(* IEC 61131-3 sources: mect_apps/TPAC1006/Collaudo_PLC, 6 files *)

(* ---- LIO_TPAC1007.gvl ---- *)
(* Global variable file *)
VAR_GLOBAL

	(* Local Input Output variables TPAC1007 *)

 	   	TP1007_LIO_Revision AT %IW5.00: UINT;

		TP1007_LIO_DigDir_1_8 AT %QB5.04: BYTE;
		TP1007_LIO_DigDir_1 AT %QX5.04.0: BOOL;
		TP1007_LIO_DigDir_2 AT %QX5.04.1: BOOL;
		TP1007_LIO_DigDir_3 AT %QX5.04.2: BOOL;
		TP1007_LIO_DigDir_4 AT %QX5.04.3: BOOL;
		TP1007_LIO_DigDir_5 AT %QX5.04.4: BOOL;
		TP1007_LIO_DigDir_6 AT %QX5.04.5: BOOL;
		TP1007_LIO_DigDir_7 AT %QX5.04.6: BOOL;
		TP1007_LIO_DigDir_8 AT %QX5.04.7: BOOL;

		TP1007_LIO_DigIn_1_8 AT %IB5.12: BYTE;
		TP1007_LIO_DigIn_1 AT %IX5.12.0: BOOL;
		TP1007_LIO_DigIn_2 AT %IX5.12.1: BOOL;
		TP1007_LIO_DigIn_3 AT %IX5.12.2: BOOL;
		TP1007_LIO_DigIn_4 AT %IX5.12.3: BOOL;
		TP1007_LIO_DigIn_5 AT %IX5.12.4: BOOL;
		TP1007_LIO_DigIn_6 AT %IX5.12.5: BOOL;
		TP1007_LIO_DigIn_7 AT %IX5.12.6: BOOL;
		TP1007_LIO_DigIn_8 AT %IX5.12.7: BOOL;

		TP1007_LIO_DigOut_1_8 AT %QB5.24: BYTE;
		TP1007_LIO_DigOut_1 AT %QX5.24.0: BOOL;
		TP1007_LIO_DigOut_2 AT %QX5.24.1: BOOL;
		TP1007_LIO_DigOut_3 AT %QX5.24.2: BOOL;
		TP1007_LIO_DigOut_4 AT %QX5.24.3: BOOL;
		TP1007_LIO_DigOut_5 AT %QX5.24.4: BOOL;
		TP1007_LIO_DigOut_6 AT %QX5.24.5: BOOL;
		TP1007_LIO_DigOut_7 AT %QX5.24.6: BOOL;
		TP1007_LIO_DigOut_8 AT %QX5.24.7: BOOL;

		TP1007_LIO_AnIn_1 AT %IW5.14: INT;
		TP1007_LIO_AnIn_2 AT %IW5.16: INT;

		TP1007_LIO_Tamb AT %IW5.18 : INT;
		TP1007_LIO_EncoderLo AT %IW5.20: UINT;
		TP1007_LIO_EncoderHi AT %IW5.22: UINT;

		TP1007_LIO_EncoderEnable AT %QW5.28: WORD;
		TP1007_LIO_EncoderReset AT %QW5.30: WORD;

		TP1007_LIO_AnOut_1 AT %QW5.26: INT;

		(* TP1007_LIO_AnIn_Conf *)
		TP1007_LIO_AnInConf_1 AT %QW5.06: WORD;
		TP1007_LIO_AnInConf_2 AT %QW5.08: WORD;

		(* TP1007_LIO_AnOut_Conf *)
		TP1007_LIO_AnOut_Conf AT %QW5.10: WORD;

		TP1007_LIO_DigIn_9_12 AT %IB5.13: BYTE;
		TP1007_LIO_DigIn_9 AT %IX5.13.0: BOOL;
		TP1007_LIO_DigIn_10 AT %IX5.13.1: BOOL;
		TP1007_LIO_DigIn_11 AT %IX5.13.2: BOOL;
		TP1007_LIO_DigIn_12 AT %IX5.13.3: BOOL;

END_VAR

(* ---- Resource1.gvl ---- *)
(* Global variable file *)
VAR_GLOBAL
RET_AnInConf_1 AT %MW0.4:UINT;
RET_AnInConf_2 AT %MW0.8:UINT;
RET_AnInConf_3 AT %MW0.12:UINT;
RET_AnInConf_4 AT %MW0.16:UINT;
RET_AnOutConf_1 AT %MW0.20:UINT;
RET_AnOutConf_2 AT %MW0.24:UINT;
CAN1_IN_DIG_8_1 AT %MW0.5380:INT;
CAN1_IN_DIG_8_2 AT %MW0.5384:INT;
CAN1_OUT_DIG_8_1 AT %MW0.5388:INT;
CAN1_OUT_DIG_8_2 AT %MW0.5392:INT;
CAN1_IN_AN_1 AT %MW0.5396:INT;
CAN1_IN_AN_2 AT %MW0.5400:INT;
CAN1_IN_AN_3 AT %MW0.5404:INT;
CAN1_IN_AN_4 AT %MW0.5408:INT;
CAN1_IN_AN_5 AT %MW0.5412:INT;
CAN1_IN_AN_6 AT %MW0.5416:INT;
CAN1_IN_AN_7 AT %MW0.5420:INT;
CAN1_IN_AN_8 AT %MW0.5424:INT;
CAN1_IN_AN_9 AT %MW0.5428:INT;
CAN1_IN_AN_10 AT %MW0.5432:INT;
CAN1_IN_AN_11 AT %MW0.5436:INT;
CAN1_IN_AN_12 AT %MW0.5440:INT;
CAN1_IN_AN_13 AT %MW0.5444:INT;
CAN1_IN_AN_14 AT %MW0.5448:INT;
CAN1_IN_AN_15 AT %MW0.5452:INT;
CAN1_IN_AN_16 AT %MW0.5456:INT;
CAN1_OUT_AN_1 AT %MW0.5460:INT;
Modbus_1 AT %MW0.5464:INT;
Parti AT %MW0.5468:INT;
END_VAR

(* ---- fb_HW119_LoadCrossTab.st ---- *)
(*[[
]]*)
FUNCTION_BLOCK fb_HW119_LoadCrossTab
#import "Resource1.gvl"
#import "crosstable.gvl"
VAR_INPUT
	ENABLE:BOOL;		(* Abilitazione funzione*)
	CTFile:STRING;		(* file di cross table da aprire	*)
	CTDimension:DINT;	(* dimensione della cross table da leggere	*)
	CTType:UINT;		(* tipo di cross table da leggere	*)
END_VAR
VAR_OUTPUT
	END:BOOL;			(* Fine funzione	*)
	ERR:BOOL;			(* segnalazione errore	*)
END_VAR
VAR
		InitXtable: fb_HW119_Init;
		ReadFields:fb_HW119_ReadVarFields;
		ReadAlarmsFields:fb_HW119_ReadAlarmsFields;
		ReadCommFields:fb_HW119_ReadCommFields;
		FBState: UINT;
		FunctRes:UINT;
		index: DINT;
		STEPS:DINT:=50;
		LowEdge:DINT:=0;
		HiEdge:DINT:=0;
END_VAR
IF ENABLE THEN
	IF FBState = 0 THEN
		InitXtable(TIPO:=CTType);													(* Inizializzazione delle variabili CT*)
		FBState:=10;
		ErrorsState:=ErrorsState AND 16#F0;											(* reset flag di errore*)
		LowEdge:=1;
		HiEdge:=STEPS;
		IF HiEdge > CTDimension THEN
			HiEdge:=CTDimension;
		END_IF;
	ELSIF FBState =10	THEN												(* OPEN CROSS TABLE*)
		FunctRes:=HW119_OpenCrossTable(CTFile);
		IF FunctRes = 0 THEN												(* Operazione andata a buon fine	*)
			FBState:=20;
			HW119_ERR[2]:=2;
		ELSE
			FBState:=1000;													(* Errore -> termina	*)
			ErrorsState:=ErrorsState OR 16#01;
			HW119_ERR[2]:=3;
		END_IF;

	ELSIF FBState =20	THEN												(* LOAD CROSS TABLE RECORDS*)
		FOR index:=LowEdge TO HiEdge	DO									(* lettura di STEPS record di CT	*)
			IF CTType > 0 	THEN											(* Se CT non è quella delle variabili non si aggiunge alla Hash*)
		 		FunctRes:=HW119_ReadCrossTableRecord(TRUE);					(* LEGGE RECORD DELLA CROSSTABLE*)
			ELSE
				FunctRes:=HW119_ReadCrossTableRecord(FALSE);				(* LEGGE RECORD DELLA CROSSTABLE lo aggiunge alla HAsh*)
			END_IF;

			IF FunctRes = 0 THEN
				HW119_ERR[1]:=2;
				CASE CTType OF
					0:		ReadFields(Index:=DINT_TO_INT(index));			(* lettura crosstable variabili	*)
							IF ReadFields.ERR THEN
								CrossTable[index].Error:=100;				(* marca la entry della crosstable come errata*)
								ErrorsState:=ErrorsState OR 16#04;
							END_IF;
					1:		ReadAlarmsFields(Index:=DINT_TO_INT(index));	(* lettura crosstable Allarmi	*)
							IF ReadAlarmsFields.ERR 	 THEN
								ALCrossTable[index].ALError:=100;			(* marca la entry della crosstable ALLARMI come errata*)
								ErrorsState:=ErrorsState OR 16#04;
							END_IF;
					ELSE
					ReadCommFields(Index:=DINT_TO_INT(index));				(* lettura CT dei parametri di comunicazione	*)
					IF index > 1 	THEN
						IF ReadCommFields.ERR 	THEN
							CommParameters[index-1].State:=FALSE;
						ELSE
							CommParameters[index-1].State:=TRUE;
						END_IF;
					 END_IF;
				END_CASE;
			ELSE
				HW119_ERR[1]:=3;
				IF CTType = 0	 THEN
					CrossTable[index].Error:=100;						(* marca la entry della crosstable come non ancora aggiornata*)
					ErrorsState:=ErrorsState OR 16#02;
				ELSIF CTType = 1	 THEN
					ALCrossTable[index].ALError:=100;					(* marca la entry della crosstable ALLARMI come non ancora aggiornata*)
					ErrorsState:=ErrorsState OR 16#04;
				END_IF;
			END_IF;

		END_FOR;
		FBState:=30;

	ELSIF FBState = 30	THEN
		LowEdge:=HiEdge+1;
		HiEdge:=HiEdge+STEPS;
		IF LowEdge < CTDimension	THEN								(* controlla se è terminata la CT da legere	*)
			IF HiEdge<CTDimension THEN
				FBState:=20;
			ELSIF HiEdge>=CTDimension THEN
				HiEdge:=CTDimension;
				FBState:=20;
			 END_IF;
		ELSE
			FBState:=40;
		END_IF;

	ELSIF FBState = 40	THEN
		FunctRes:=HW119_CloseCrossTable();											(* CLOSE CrossTable*)
		IF FunctRes = 0 THEN
			HW119_ERR[0]:=2;				(*debug*)
		 	FBState:= 100;
		ELSE
			FBState:=1000;
			HW119_ERR[0]:=3;				(*debug*)
			ErrorsState:=ErrorsState OR 16#08;
		END_IF;
	ELSIF FBState = 100	THEN														(* TERMINATA LETTURA CROSSTABLE*)
		END:=TRUE;
	ELSIF FBState = 1000 THEN														(* TERMINATA LETTURA CROSSTABLE*)
		FunctRes:=HW119_CloseCrossTable();											(* CLOSE CrossTable*)
		FBState:= 1010;
		ERR:=TRUE;
	END_IF;
ELSE
	END:=FALSE;
	ERR:=FALSE;
	FBState:= 0;
END_IF;
END_FUNCTION_BLOCK

(* ---- fb_HW119_ReadAlarmsFields.st ---- *)
(*[[
]]*)
FUNCTION_BLOCK fb_HW119_ReadAlarmsFields
#import "Resource1.gvl"
#import "crosstable.gvl"
VAR_INPUT
	Index:INT;
END_VAR
VAR_OUTPUT
	ERR:BOOL;
END_VAR

VAR
	Field:STRING;
	FunctRes:UINT;
END_VAR

	ERR:=FALSE;
	FunctRes:=HW119_GetCrossTableField(Field);				(*Lettura TIPO 0 : evento, 1 : allarme*)
	IF FunctRes = 0 THEN
		ALCrossTable[index].ALType:=STRING_TO_BOOL(Field);
	ELSE
		ERR:=TRUE;
	END_IF;

	FunctRes:=HW119_GetCrossTableField(Field);				(* variabile di allarme	*)
	IF FunctRes = 0 THEN
		ALCrossTable[index].ALTag:=Field;
	ELSE
		ERR:=TRUE;
	END_IF;

	FunctRes:=HW119_GetCrossTableField(Field);				(* Variabile di sorgente	*)
	IF FunctRes = 0 THEN
		ALCrossTable[index].ALSource:=Field;
	ELSE
		ERR:=TRUE;
	END_IF;

	FunctRes:=HW119_GetCrossTableField(Field);				(* variabile di confronto	*)
	IF FunctRes = 0 THEN
		ALCrossTable[index].ALCompareVar:=Field;
	ELSE
		ERR:=TRUE;
	END_IF;

	FunctRes:=HW119_GetCrossTableField(Field);
	IF FunctRes = 0 THEN
		ALCrossTable[index].ALCompareVal:=STRING_TO_DWORD(Field);
	ELSE
		ERR:=TRUE;
	END_IF;

	FunctRes:=HW119_GetCrossTableField(Field);
	IF FunctRes = 0 THEN
		ALCrossTable[index].ALOperator:=STRING_TO_UINT(Field);
	ELSE
		ERR:=TRUE;
	END_IF;

	FunctRes:=HW119_GetCrossTableField(Field);
	IF FunctRes = 0 THEN
		ALCrossTable[index].ALFilterTime:=STRING_TO_UINT(Field);
		ALCrossTable[Index].ALFilterCount:=ALCrossTable[index].ALFilterTime;
	ELSE
		ERR:=TRUE;
	END_IF;

END_FUNCTION_BLOCK

(* ---- PLC.st ---- *)
(*[[
]]*)
PROGRAM PLC
#import "Resource1.gvl"
#import "crosstable.gvl"
#import "TPACLocaIO.gvl" (* <---= *)
#import "Collaudo_CAN.gvl"
#import "LIO_TPAC1006.gvl"
VAR
	fb_HW119_PLCwriteVar_Inst : fb_HW119_PLCwriteVar;
	counter : UDINT := 0;
	divisor : UDINT := 10;
	values : ARRAY [0..15] OF DWORD;
	TIMER1:TON;
	TIMER2:TON;
END_VAR;
if Parti = 1 then
	TIMER2(IN:=TRUE,PT:=T#1s);
	IF TIMER2.Q THEN
	TIMER2(IN:=FALSE,PT:=T#1s);
		if counter = 0 * divisor then
			PLC_DigOut_1:=0;
			PLC_DigOut_2:=0;
			PLC_DigOut_3:=0;
			PLC_DigOut_4:=0;
			PLC_DigOut_5:=0;
			PLC_DigOut_6:=0;
			PLC_DigOut_7:=0;
			PLC_DigOut_8:=0;
			PLC_DigOut_9:=0;
			PLC_DigOut_10:=0;
			PLC_DigOut_11:=0;
			PLC_DigOut_12:=0;
			PLC_DigOut_13:=0;
			PLC_DigOut_14:=0;
			PLC_DigOut_15:=0;
			PLC_DigOut_16:=0;
		elsif counter = 1  then
			PLC_DigOut_1 := 1;
		elsif counter = 2  then
			PLC_DigOut_1 := 0;
			PLC_DigOut_2 := 1;
		elsif counter = 3 then
			PLC_DigOut_2 := 0;
			PLC_DigOut_3 := 1;
		elsif counter = 4 then
			PLC_DigOut_3 := 0;
			PLC_DigOut_4 := 1;
		elsif counter = 5 then
			PLC_DigOut_4 := 0;
			PLC_DigOut_5 := 1;
		elsif counter = 6 then
			PLC_DigOut_5 := 0;
			PLC_DigOut_6 := 1;
		elsif counter = 7 then
			PLC_DigOut_6 := 0;
			PLC_DigOut_7 := 1;
		elsif counter = 8 then
			PLC_DigOut_7 := 0;
			PLC_DigOut_8 := 1;
		elsif counter = 9 then
			PLC_DigOut_8 := 0;
			PLC_DigOut_9 := 1;
		elsif counter = 10 then
			PLC_DigOut_9 := 0;
			PLC_DigOut_10 := 1;
		elsif counter = 11 then
			PLC_DigOut_10 := 0;
			PLC_DigOut_11 := 1;
		elsif counter = 12  then
			PLC_DigOut_11 := 0;
			PLC_DigOut_12 := 1;
		end_if;

		counter := counter + 1;

		if counter > 13  then
			counter := 0;
		end_if;
	end_if;

values[0]:=1;
fb_HW119_PLCwriteVar_Inst(VARIABLE := 'Modbus_1', VALUES := values, Nregs := 1);
IF FALSE THEN
	ch1_CAN1_OUT_DIG_8_1:=0;
END_IF;
TIMER1(in:=TRUE,PT:=T#1s);
IF TIMER1.Q THEN
	TIMER1(in:=FALSE,PT:=T#1s);
	IF ch1_CAN1_OUT_DIG_8_1 = 16#01 THEN
		ch1_CAN1_OUT_DIG_8_1:=16#01;
	ELSE
		ch1_CAN1_OUT_DIG_8_1:=16#00;
	END_IF;
END_IF;
end_if;
PLC_CAN1_IN_AN_1:=ch1_CAN1_IN_AN_1;
PLC_CAN1_IN_AN_2:=ch1_CAN1_IN_AN_2;
PLC_CAN1_IN_AN_3:=ch1_CAN1_IN_AN_3;
PLC_CAN1_IN_AN_4:=ch1_CAN1_IN_AN_4;
PLC_CAN1_IN_AN_5:=ch1_CAN1_IN_AN_5;
PLC_CAN1_IN_AN_6:=ch1_CAN1_IN_AN_6;
PLC_CAN1_IN_AN_7:=ch1_CAN1_IN_AN_7;
PLC_CAN1_IN_AN_8:=ch1_CAN1_IN_AN_8;
PLC_CAN1_IN_AN_9:=ch1_CAN1_IN_AN_9;
PLC_CAN1_IN_AN_10:=ch1_CAN1_IN_AN_10;
PLC_CAN1_IN_AN_11:=ch1_CAN1_IN_AN_11;
PLC_CAN1_IN_AN_12:=ch1_CAN1_IN_AN_12;
PLC_CAN1_IN_AN_13:=ch1_CAN1_IN_AN_13;
PLC_CAN1_IN_AN_14:=ch1_CAN1_IN_AN_14;
PLC_CAN1_IN_AN_15:=ch1_CAN1_IN_AN_15;
PLC_CAN1_IN_AN_16:=ch1_CAN1_IN_AN_16;
if  PLC_AnOutConf_1 <> UINT_TO_WORD(RET_AnOutConf_1)then
	PLC_AnOut_1 := 0;
	PLC_AnOutConf_1 := UINT_TO_WORD(RET_AnOutConf_1);
end_if;
if  PLC_AnOutConf_2 <> UINT_TO_WORD(RET_AnOutConf_2)then
	PLC_AnOut_2 := 0;
	PLC_AnOutConf_2 := UINT_TO_WORD(RET_AnOutConf_2);
end_if;

PLC_AnInConf_1 := UINT_TO_WORD(RET_AnInConf_1);
PLC_AnInConf_2 := UINT_TO_WORD(RET_AnInConf_2);
PLC_AnInConf_3 := UINT_TO_WORD(RET_AnInConf_3);
PLC_AnInConf_4 := UINT_TO_WORD(RET_AnInConf_4);

(* limits the overflow value *)
IF (INT_TO_WORD(TP1006_LIO_AnOut_Conf) AND 16#01) = 16#01 THEN
	IF PLC_AnOut_1 > 2000 then
		PLC_AnOut_1:=2000;
	END_IF;
	IF PLC_AnOut_1 < 0 then
		PLC_AnOut_1:=0;
	END_IF;
END_IF;
IF (INT_TO_WORD(TP1006_LIO_AnOut_Conf) AND 16#02) = 16#02 THEN
	IF PLC_AnOut_1 > 1000 then
		PLC_AnOut_1:=1000;
	END_IF;
	IF PLC_AnOut_1 < 0 then
		PLC_AnOut_1:=0;
	END_IF;
END_IF;
IF (INT_TO_WORD(TP1006_LIO_AnOut_Conf) AND 16#10)  = 16#10 THEN
	IF PLC_AnOut_2 > 2000 then
		PLC_AnOut_2:=2000;
	END_IF;
	IF PLC_AnOut_2 < 0 then
		PLC_AnOut_2:=0;
	END_IF;
END_IF;
IF (INT_TO_WORD(TP1006_LIO_AnOut_Conf) AND 16#20)  = 16#20 THEN
	IF PLC_AnOut_2 > 1000 then
		PLC_AnOut_2:=1000;
	END_IF;
	IF PLC_AnOut_2 < 0 then
		PLC_AnOut_2:=0;
	END_IF;
END_IF;
END_PROGRAM

(* ---- Program1.st ---- *)
(*[[
    UserHelpURL= "4cfile:Program1.HTML",
]]*)

PROGRAM Program1
#import "crosstable.gvl"
VAR
(* Revisione 5.31
Corretto baco nel blocco funzione PLCsync
riga 35					FOR I:=0 TO CrossTable[addr].NReg-1 BY STEPS DO
aggiunto -1 al FOR
*)

(* Revisione 5.32
Inserita la misurazione della query pause al termine della risposta dallo slave
solo per protocollo RTU
*)

(* Revisione 5.33
Modificata policy del device disconnesso. Ora, se un indirizzo non risponde e supera il limite faildivisor
si mette l'indirizzo in una blacklist, quindi le richieste di accessi successivi al device saranno ignorati

Revisione 5.4
Inseriti contatori di errori per ogni protocollo
	ContatoreErroriRTU
	ContatoreErroriTCP
	ContatoreErroriTCPRTU

Inserite variabili di revisione:
	PLCRevision01
	PLCRevision02

Modificata scrittura in uPLC: Le scritture sono prioritarie rispetto a quelle HMI, sono ammesse le scritture multiple
Inserita la gestione delle variabili intere a 32 bit
	UDINTDCBA
	UDINTCDAB
	UDINTABCD
	UDINTBADC
	DINTDCBA
	DINTCDAB
	DINTABCD
	DINTBADC

 Revisione 5.42
 	Inserite scritture ad alta priorità da uPLC
	Le scritture sono inserite in tre code (una per protocollo) ed eseguite nella sequenza di arrivo
	tutte le altre operazioni sono ritardate fino a che non sono
	terminate le scritture

Revisione 5.43
	Corretto baco già risolto in 5.31, reintrodotto nella 5.4.
Revisione 5.44
	Corretto baco sulla gestione allarmi: Non veniva effettuato l'aggiornamento dello stato della variabile a error=0
		nel caso di accessi interni (non su strumenti) sia da HMI che da uPLC
		Perciò se la SourceVariable era una variabile interna (non su un device modbus)
		non veniva aggiornato lo stato di variabile disponibile per gli allarmi
		corretto file PLC_sync.st
		aggiunta alla riga 35 CrossTable[addr+I].Error:=0;
	Corretto baco sulle scritture da PLC:
		non venivano effettuate le scritture multiple se il uPLC le effettuava su variabili interne
		modificato nel blocco funzione fb_HW119_PLCwriteVar il codice
					FOR I:=0 TO NRegs-1 DO
						ARRAY_CROSSTABLE_INPUT[WORD_TO_INT(ADDRESS)+I]:=CrossTable[WORD_TO_INT(ADDRESS)+I].PLCWriteVal;
						CrossTable[WORD_TO_INT(ADDRESS)+I].Error:=0;
					END_FOR;
Revisione 5.45
	Corretto baco su scritture multiple

Revisione 5.46
	Corretto baco su scritture singole

Revisione 5.47
	Modificata gestione ricetta
	Aggiunta scrittura in ricetta delle variabili interne

Revisione 5.48
	Corretta la gestione dei falg di busywrite per le scritture su variabili interne nel blocco funzione PLCsync
Revisione 5.49
	Corretto baco su FB plcsync: non veniva aggiornata la mandata in run del protocollo TCP a seguito di una riconnessione
Revisione 5.50
	Corretta letura Modbus sui bit nei protocolli RTU e TCPRTU
Revisione 5.51
	Corretta la gestione della scrittura a bit da PLC interno
	Corretta la segnalazione di errore nel blocco funzione fb_HW119_PLCwriteVar
	MOdificato blocco fb_HW119_AlarmsMngr: in caso di variabili interne non si controlla se è già avvenuta l'assegnazione
Revisione 5.52
	Corretta gestione fb_HW119_PLCwritevar in caso di errore sulla funzione Gettaddr()
Revisione 5.53
	Aggiunta scrittura multipla delle variabili interne
Revisione 6.00
	Inserita priorità delle letture
	contatori errore e blacklist
	scritture ad interrupt
Revisione 6.01
	Corretti bachi:
		La variabile Retry non veniuva azzerata se il dispositivo ritornava on line prima dello scadere dei retry
		messa a false la variabile debug
		corretta la revisione sw
		aggiunta variabilie di Error_flag che segnala se c'è stato almeno un errore dall'ultimo reset
Revisione 6.02
		corretto baco su scrittura da PLC
		aggiunto a Error_flag la segnalazione di errore sulla lettura di una crosstable
Revisione 6.03
		modificate costanti dei file delle CT: tolti i path per poter essere utilizzati da SD
		non si tiene conto del  path per le crosstable per il caricamento da Flash o SD card
Revisione 6.04
	Inserito di default NodeId a 1 nel caso di protocollo TCP

Revisione 6.05
	Inserita gestione Canopen in funzione della variabile HardwareType
	variata la gestione delle scritture e letture nel task RTU
Revisione 6.08
	corretti bachi sui protocolli
Revisione 6.10
	corretti bacho su fb_HW119_MODBUS
Revisione 6.12
	Modificati file gvl delle variabili locali
	creato blocco funzione di sincronizzazione per le variabili locali del tpac1007
	unificate le variabili di IO locale PLC di accesso utente
	inserita la variabile di sistema PLC_time per che si azzera ogni 3600 secondi
 Revisione 6.13
 	Modificate uscite analogiche sui blocchi funzione fb_TPAC1006_LIO_sync e fb_TPAC1007_LIO_sync
*)

	InitComm:fb_HW119_InitComm;
	AlarmMngr:fb_HW119_AlarmsMngr;
	LoadXTable:fb_HW119_LoadCrossTab;
	ErrorMNG:fb_HW119_ErrorMng;
	PLCsync:fb_HW119_PLCsync;
	Reconnect:fb_HW119_Check;
	TPAC1006_LIOsync:fb_TPAC1006_LIOsync;
	TPAC1007_LIOsync:fb_TPAC1007_LIOsync;
	TICtimer:fb_TPAC_tic;
	FunctRes:UINT;
	CommState: UDINT;
	COUNTER:UDINT;
	timer_sync:TON;

	(* DEBUG
	errorT1:DINT;
	errorT2:DINT;
	errorT3:DINT;
	errorT4:DINT;
	reterr:WORD;
	*)
END_VAR
(*	DEBUG
	errorT1:=GetLocalTaskErrno ('Task1');
	errorT2:=GetLocalTaskErrno ('Task2_RTU'	);
	errorT3:=GetLocalTaskState ('Task1');
	errorT4:=GetLocalTaskState('Task2_RTU');
	PLCRevision01:=5;
	PLCRevision02:=4;
*)

	IF CommState = 0	THEN
		FunctRes:=HW119_CloseCrossTable();
		LoadXTable(ENABLE:=FALSE);
		InitComm(ENABLE:=FALSE);
		ErrorsState:=0;
		CommState:=10;
		COUNTER:=0;
		RTU_RUN:=FALSE;
		TCP_RUN:=FALSE;
		TCPRTU_RUN:=FALSE;
		ERROR_FLAG:=0;
	ELSIF CommState = 10	THEN			(* Lettura crosstable allarmi	*)
		LoadXTable(ENABLE:=TRUE,CTFile:=ALcrossTableFile,CTDimension:=DimAlarmsCT,CTType:=1);
		IF LoadXTable.ERR  	THEN
			CommState:=20;					(* Fallita lettura crosstable allrmi -> prosegue con lettura cross table variabili*)
			ALCrossTableState:=FALSE;
			LoadXTable(ENABLE:=FALSE);
			ERROR_FLAG:=ERROR_FLAG OR 16#10;(* SEGNALO L'ERRORE SUL BIT 4*)
		ELSE
			IF LoadXTable.END THEN
				CommState:=20;				(*lettura crosstable  Allarmi  OK  -> prosegue*)
				FunctRes:=HW119_CloseCrossTable();
				LoadXTable(ENABLE:=FALSE);
			END_IF;
		END_IF;

	ELSIF CommState = 20	THEN			(* Lettura crosstable variabili	*)
		LoadXTable(ENABLE:=TRUE,CTFile:=VARcrossTableFile,CTDimension:=DimCrossTable,CTType:=0);
		IF LoadXTable.ERR  	THEN
			CommState:=1000;
			CrossTableState:=FALSE;			(* Fallita lettura crosstable  variabili: FINE*)
			ERROR_FLAG:=ERROR_FLAG OR 16#20;(* SEGNALO L'ERRORE SUL BIT 5*)
		ELSE
			IF LoadXTable.END THEN
				CommState:=30;				(*lettura crosstable  variabili  OK ->  prosegue*)
				LoadXTable(ENABLE:=FALSE);
			END_IF;
		END_IF;

	ELSIF CommState = 30	THEN			(* Lettura crosstable parametri di comunicazione	*)
		LoadXTable(ENABLE:=TRUE,CTFile:=CommParFile,CTDimension:=5,CTType:=2);
		IF LoadXTable.ERR  	THEN
			CommState:=1000;				(* Fallita lettura crosstable  parametri di comunicazione: FINE*)
			ERROR_FLAG:=ERROR_FLAG OR 16#08;(* SEGNALO L'ERRORE SUL BIT 3*)
		ELSE
			IF LoadXTable.END THEN
				CommState:=40;				(*lettura crosstable  variabili  OK ->  prosegue*)
				LoadXTable(ENABLE:=FALSE);
			END_IF;
		END_IF;

	(* Abilitazione protocollo RTU se almeno una entry della crosstable supporta questo protocollo*)
	ELSIF CommState = 40	THEN
		IF 	RTUProtocol_ON	AND CommParameters[1].State THEN
			InitComm(ENABLE:=TRUE,Interface:='RTU');	(*inizializza comunicazione	*)
			IF InitComm.END THEN
				FunctRes:=WORD_TO_UINT(TSK_Start('TASK2_RTU'));		(* partenza task RTU*)
				ERROR_FLAG:=ERROR_FLAG OR 16#80;(* SEGNALO CHE IL TASK RTU è PARTITO*)
				CommState:=50;
				InitComm(ENABLE:=FALSE);
				RTU_RUN:=TRUE;
			ELSIF InitComm.ERR THEN
				CommState:=50;
				InitComm(ENABLE:=FALSE);
				RTU_RUN:=FALSE;
			END_IF;
		ELSE
			CommState:=50;
		END_IF;

	(* Abilitazione protocollo TCP se almeno una entry della crosstable supporta questo protocollo*)
	ELSIF CommState = 50	THEN
		IF 	TCPProtocol_ON	AND CommParameters[2].State THEN
			InitComm(ENABLE:=TRUE,Interface:='TCP');	(*inizializza comunicazione	*)
			IF InitComm.END THEN
				FunctRes:=WORD_TO_UINT(TSK_Start('TASK3_TCP'));		(* partenza task TCP*)
				ERROR_FLAG:=ERROR_FLAG OR 16#100;(* SEGNALO CHE IL TASK TCP è PARTITO*)
				CommState:=60;
				InitComm(ENABLE:=FALSE);
				TCP_RUN:=TRUE;
			ELSIF InitComm.ERR THEN
				CommState:=60;
				InitComm(ENABLE:=FALSE);
				TCP_RUN:=FALSE;
			END_IF;
		ELSE
			CommState:=60;
		END_IF;

	(* Abilitazione protocollo TCPRTU se almeno una entry della crosstable supporta questo protocollo*)
	ELSIF CommState = 60 	THEN

		IF 	TCPRTUProtocol_ON	AND CommParameters[3].State THEN
			InitComm(ENABLE:=TRUE,Interface:='TCPRTU');	(*inizializza comunicazione	*)
			IF InitComm.END THEN
				FunctRes:=WORD_TO_UINT(TSK_Start('TASK4_TCPRTU'));		(* partenza task TCPRTU*)
				ERROR_FLAG:=ERROR_FLAG OR 16#200;(* SEGNALO CHE IL TASK TCPRTU è PARTITO*)
				CommState:=70;
				InitComm(ENABLE:=FALSE);
				TCPRTU_RUN:=TRUE;
			ELSIF InitComm.ERR THEN
				TCPRTU_RUN:=FALSE;
				CommState:=70;
				InitComm(ENABLE:=FALSE);
			END_IF;
		ELSE
			CommState:=70;
		END_IF;

	ELSIF CommState = 70	THEN
		ERROR_FLAG:=ERROR_FLAG OR 16#40;	(* SEGNALA SUL BIT 6 CHE HA TERMINATO L'INIZIALIZZAZIONE DELLE CT*)
		TRIGGER02:=TRIGGER02;
		TRIGGER01:=TRIGGER01;
		IF  ALCrossTableState THEN
			CommEnabled:=TRUE;
		END_IF;
		FunctRes:=WORD_TO_UINT(TSK_Start('TASK0_Control'));		(* partenza task PLC*)
		CommState:=80;

	ELSIF CommState = 80	THEN
		TRIGGER02:=TRIGGER02;
		TRIGGER01:=TRIGGER01;
		IF CommEnabled THEN
			AlarmMngr();					(* Gestione allarmi*)
		END_IF;
		Reconnect();						(* Riconnessione per protocolli TCP e TCPRTU	*)
		PLCsync();							(* sincronizzazione tra variabili PLC e HMI	*)
		timer_sync(IN:=TRUE,PT:=T#50ms);
		IF timer_sync.Q THEN
			timer_sync(IN:=FALSE);
			TICtimer(tic:=T#50ms);
			IF (HardwareType AND 16#000000FF) >= 16#01 THEN
				TPAC1006_LIOsync();
			END_IF;
			IF (HardwareType AND 16#00FF0000) >= 16#01 THEN
				TPAC1007_LIOsync();
			END_IF;
		END_IF;
	ELSIF CommState = 1000	THEN
		TRIGGER02:=TRIGGER02;
		ERROR_FLAG:=ERROR_FLAG OR 16#40;	(* SEGNALA SUL BIT 6 CHE HA TERMINATO L'INIZIALIZZAZIONE DELLE CT*)
		ErrorMNG();							(* Gestione errori	*)
	END_IF;
END_PROGRAM
